FUNCTION_BLOCK PrintStation EXTENDS MultiStation
VAR_INPUT
	StationEnable: ARRAY[0..GVL.PRINT_NUM_STATIONS - 1] OF BOOL;
END_VAR
VAR_OUTPUT
	MoversInPosition: BOOL;
END_VAR
VAR
END_VAR

METHOD Cyclic : BOOL
VAR
	i : USINT;
	Init: BOOL;
END_VAR
// Initializations
IF NOT Init THEN
;
END_IF

// Detect New Movers
IF PositionTrigger.MoverPassedPosition THEN
	FOR i := GVL.PRINT_NUM_STATIONS - 1 TO 0 BY -1 DO
		IF StationEnable[i] AND NOT Station[i].TrackedMoverCount < 0 THEN
			PositionTrigger.CurrentMover.MoveToStation(Station[i]);
			EXIT;
		END_IF
	END_FOR
END_IF

// Determine if all movers are in position
MoversInPosition	:= TRUE;
FOR i := 0 TO GVL.PRINT_NUM_STATIONS - 1 DO
	IF (Station[i].TrackedMoverCount <> 1) THEN	MoversInPosition := FALSE; EXIT;
	ELSIF Station[i].TrackedMoverCount = 1 THEN
		IF Station[i].CurrentMover.CurrentMoveType = MOVETYPE_NONE THEN MoversInPosition := FALSE; EXIT; END_IF
	END_IF
END_FOR

// Call Cyclics
PositionTrigger.Cyclic();
FOR i := 0 TO GVL.PRINT_NUM_STATIONS - 1 DO
	IF StationEnable[i] THEN
		Station[i].Cyclic();
	END_IF
END_FOR
END_METHOD

END_FUNCTION_BLOCK

(* stored: Version 1.1.0.1, ProductVersion 3.1.4024.12
   POU PrintStation: Id {af37668e-bf92-0c4b-10be-9a89eaacc2a8}, SpecialFunc None
   Folder Methods: Id {932d410e-fce3-0267-2e8d-d5af7357858b}
   Folder Properties: Id {6c126d4c-4a9b-0de2-06e7-ed27335d9ce3}
   Method Cyclic: Id {a16d672c-6e58-0f87-0490-601abb6d509d} *)
